TYPE UR_6_T2O_IntRegisters :
STRUCT
		Ints:ARRAY[0..23] OF DINT;
END_STRUCT
END_TYPE

(* stored: Version 1.1.0.1
   DUT UR_6_T2O_IntRegisters: Id {90d3bb7a-b510-4654-a25b-2f60d5a91d8d} *)
